FUNCTION_BLOCK HOME_RUN
VAR_INPUT
END_VAR
VAR_OUTPUT
END_VAR
VAR
END_VAR

END_FUNCTION_BLOCK

(* stored: Version 1.1.0.1, ProductVersion 3.1.4022.18
   POU HOME_RUN: Id {14f79e0e-6d78-4dd0-b34b-643ee51b376d}, SpecialFunc None *)
